// TIA Portal V19 export
DATA_BLOCK "PW TRANSFER PUMP"   // DB14
{ S7_Optimized_Access := 'TRUE' }
// stored: MemoryReserve 100
   VAR
      "TRASNFER START/STOP" : Bool;
   END_VAR
BEGIN
END_DATA_BLOCK
